// TIA Portal project "Cvik2" (V16)
// Bobrov, Boltian

(* hardware
DEVICE "S7-1200 station_2"  S7-1200 Station
   slot 0: "Rack_0"  S7-1200 Rack  Rack  V1.0
   slot 1: "PLC_6"  CPU 1215C DC/DC/DC  6ES7 215-1AG40-0XB0  V4.4
*)

// ===== PLC "PLC_6"  CPU 1215C DC/DC/DC =====

VAR_GLOBAL   // PLC tag table "Default tag table"
   "os1" AT %I0.0 : Bool;
   "os2" AT %I0.1 : Bool;
   "Direction" AT %Q0.0 : Bool;
   "Direction_1" AT %Q0.1 : Bool;
   "Mode 0" AT %M0.2 : Bool;
   "Mode 1" AT %M0.3 : Bool;
   "Mode 2" AT %M0.4 : Bool;
   "Smer" AT %MW8 : Int;
   "Mode" AT %MW6 : Int;
   "CONTROL BIT  M1" AT %M0.7 : Bool;
END_VAR

ORGANIZATION_BLOCK "Main"   // OB1, LAD, ProgramCycle
TITLE = "Main Program Sweep (Cycle)"
{ S7_Optimized_Access := 'TRUE' }
VERSION : 0.1
   VAR_INPUT
      Initial_Call : Bool;   // Initial call of this OB
      Remanence : Bool;   // =True, if remanent data are available
   END_VAR
   VAR_TEMP   // added for the SCL form of the ladder/FBD networks
      _w1 : Bool;
   END_VAR
BEGIN

REGION Network 1
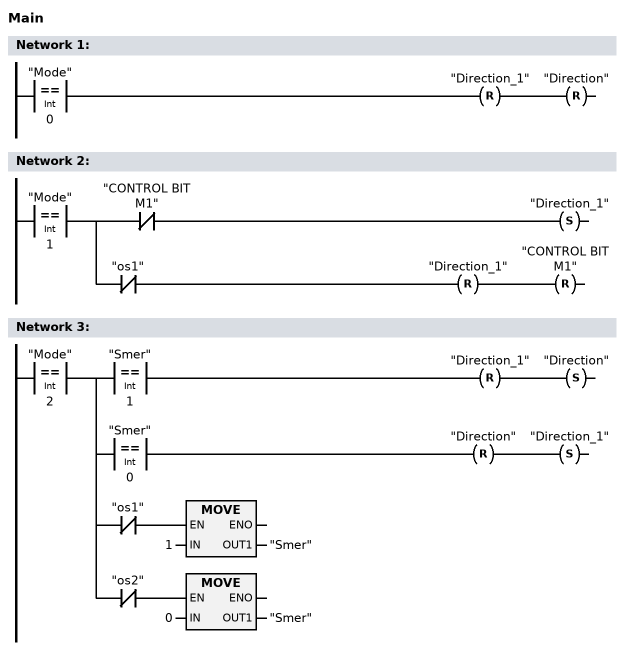
   RUNG wire#powerrail
      { S7_Templates := "SrcType := Int" } EQ_Contact(in1 := "Mode", in2 := 0)
      R_Coil( "Direction_1" )
      R_Coil( "Direction" )
   END_RUNG
   // the same network as SCL:
   IF "Mode" = 0 THEN
       "Direction_1" := FALSE;
       "Direction" := FALSE;
   END_IF;
END_REGION

REGION Network 2
   RUNG wire#powerrail
      { S7_Templates := "SrcType := Int" } EQ_Contact(in1 := "Mode", in2 := 1)
      wire#w1
      I_Contact( "CONTROL BIT  M1" )
      S_Coil( "Direction_1" )
   END_RUNG
   RUNG wire#w1
      I_Contact( "os1" )
      R_Coil( "Direction_1" )
      R_Coil( "CONTROL BIT  M1" )
   END_RUNG
   // the same network as SCL:
   #_w1 := "Mode" = 1;
   IF #_w1 AND NOT "CONTROL BIT  M1" THEN "Direction_1" := TRUE; END_IF;
   IF #_w1 AND NOT "os1" THEN
       "Direction_1" := FALSE;
       "CONTROL BIT  M1" := FALSE;
   END_IF;
END_REGION

REGION Network 3
   RUNG wire#powerrail
      { S7_Templates := "SrcType := Int" } EQ_Contact(in1 := "Mode", in2 := 2)
      wire#w1
      { S7_Templates := "SrcType := Int" } EQ_Contact(in1 := "Smer", in2 := 1)
      R_Coil( "Direction_1" )
      S_Coil( "Direction" )
   END_RUNG
   RUNG wire#w1
      { S7_Templates := "SrcType := Int" } EQ_Contact(in1 := "Smer", in2 := 0)
      R_Coil( "Direction" )
      S_Coil( "Direction_1" )
   END_RUNG
   RUNG wire#w1
      I_Contact( "os1" )
      Move(in := 1, out1 => "Smer")
   END_RUNG
   RUNG wire#w1
      I_Contact( "os2" )
      Move(in := 0, out1 => "Smer")
   END_RUNG
   // the same network as SCL:
   #_w1 := "Mode" = 2;
   IF #_w1 AND ("Smer" = 1) THEN
       "Direction_1" := FALSE;
       "Direction" := TRUE;
   END_IF;
   IF #_w1 AND ("Smer" = 0) THEN
       "Direction" := FALSE;
       "Direction_1" := TRUE;
   END_IF;
   IF #_w1 AND NOT "os1" THEN "Smer" := 1; END_IF;
   IF #_w1 AND NOT "os2" THEN "Smer" := 0; END_IF;
END_REGION
END_ORGANIZATION_BLOCK